{attribute 'pack_mode' := '2'}
TYPE ST_CTRL_NCI :
STRUCT
  eCmd        : E_NCI_CTRL := E_NCI_CTRL.INIT;
  rOverride   : REAL := 47.11;

END_STRUCT
END_TYPE

(* stored: Version 1.1.0.1, ProductVersion 3.1.4024.12
   DUT ST_CTRL_NCI: Id {409f0024-413b-084a-0caa-73fd90ffc9ad} *)
